// TIA Portal V18 export
DATA_BLOCK "System_Enable_DB"   // DB15
// stored: AutoNumber false, InstanceOfName System_Enable, InstanceOfType FB
"System_Enable"
BEGIN
END_DATA_BLOCK
